TYPE EM_Transport_Mechanische_Stop_HMI :
STRUCT
	Start		: BOOL;
	Stop		: BOOL;
	Reset		: BOOL;
	Abort		: BOOL;
	Auto		: BOOL;
	Manueel		: BOOL;
END_STRUCT
END_TYPE

(* stored: Version 1.1.0.1, ProductVersion 3.1.4024.12
   DUT EM_Transport_Mechanische_Stop_HMI: Id {2bd21dc5-0fd2-4e09-b68d-3aa0e8c6e9f4} *)
